FUNCTION_BLOCK FB_FMS205_Producir_SFC
VAR_INPUT
	Producir: BOOL;
END_VAR
VAR_OUTPUT
END_VAR

VAR_IN_OUT
	mdAlimentador: FB_Alimentador;	
	mdPickAndPlaceCarga: FB_PickAndPlace;
END_VAR

VAR
END_VAR

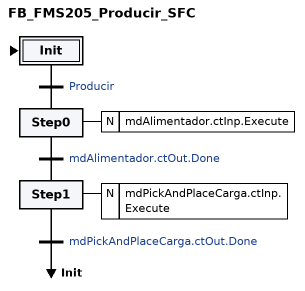
INITIAL_STEP Init:
END_STEP
TRANSITION FROM Init TO Step0
    := Producir;
END_TRANSITION
STEP Step0:
    mdAlimentador.ctInp.Execute(N);
END_STEP
TRANSITION FROM Step0 TO Step1
    := mdAlimentador.ctOut.Done;
END_TRANSITION
STEP Step1:
    mdPickAndPlaceCarga.ctInp.Execute(N);
END_STEP
TRANSITION FROM Step1 TO Init
    := mdPickAndPlaceCarga.ctOut.Done;
END_TRANSITION

END_FUNCTION_BLOCK

(* stored: Version 1.1.0.1, ProductVersion 3.1.4024.11
   POU FB_FMS205_Producir_SFC: Id {a81c472c-1220-4b76-860b-f7f6b111694f}, SpecialFunc None *)
